FUNCTION_BLOCK BasicTest (* Template for a simple Basic Function Block Type *)
  (* Standard: 61499-2 *)
  (* Version 1.0, 2019-04-02, michael *)
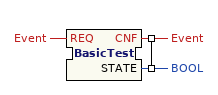
  EVENT_INPUT
    REQ; (* Normal Execution Request *)
  END_EVENT
  EVENT_OUTPUT
    CNF WITH STATE; (* Execution Confirmation *)
  END_EVENT
  VAR_OUTPUT
    STATE : BOOL; (* Output event qualifier *)
  END_VAR
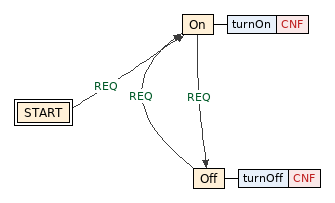
  EC_STATES
    START; (* Initial State *)
    On : turnOn -> CNF;
    Off : turnOff -> CNF;
  END_STATES
  EC_TRANSITIONS
    START TO On := REQ;
    On TO Off := REQ;
    Off TO On := REQ;
  END_TRANSITIONS
  ALGORITHM turnOn IN ST: (* new algorithm *)
STATE := TRUE;
  END_ALGORITHM
  ALGORITHM turnOff IN ST: (* new algorithm *)
STATE:=FALSE;
  END_ALGORITHM
END_FUNCTION_BLOCK
